Staubli VAL3: displayMenu.pgx

public program displayMenu(string x_sMenu)
  local string l_sMenuItm[8]
  local num l_i
begin
  // This routine displays a menu on the last line of the teach pendant
  // and wait until the user selects one of the item of the menu.
  //
  // Input Param
  //  x_sItem : Menu to be displayed
  //
  // Output param
  //  xSelect : Number of the selected item in range of 1 to 8
  //
  // Created 23-02-05                           C.CURRIVAND
  //------------------------------------------------------------------
  // Convertion
  call _str2Array(x_sMenu," ",l_sMenuItm)
  for l_i=0 to 7
    if l_sMenuItm[l_i]!=""
      call typeMenu(l_i+1,l_sMenuItm[l_i])
    endIf
  endFor
end
